PROGRAM MotionControl_sfc
VAR
	mcPower : MC_Power;
	mcSetPosition: MC_SetPosition;
	mcMoveAboslute: MC_MoveAbsolute;
	mcMoveRelative: MC_MoveRelative;
	mcMoveVelocity: MC_MoveVelocity;
	mcReset:MC_Reset;
	mcHalt:MC_Halt;
	mcStop:MC_Stop;
	
	bEnable : BOOL;
	bExecute_SPOS :BOOL;
	bExecute_MABS :BOOL;
	bExecute_MREL :BOOL;
	bExecute_RES :BOOL;
	bExecute_VEL :BOOL;
	bExecute_HALT :BOOL;
	bExecute_STOP :BOOL;
	
	fVelocity:LREAL;
	fPosition:LREAL;
	
	
	fAccel:LREAL;
END_VAR
VAR // added by the converter: edge detectors and wires of the graphical bodies
    _w1 : ANY;
END_VAR

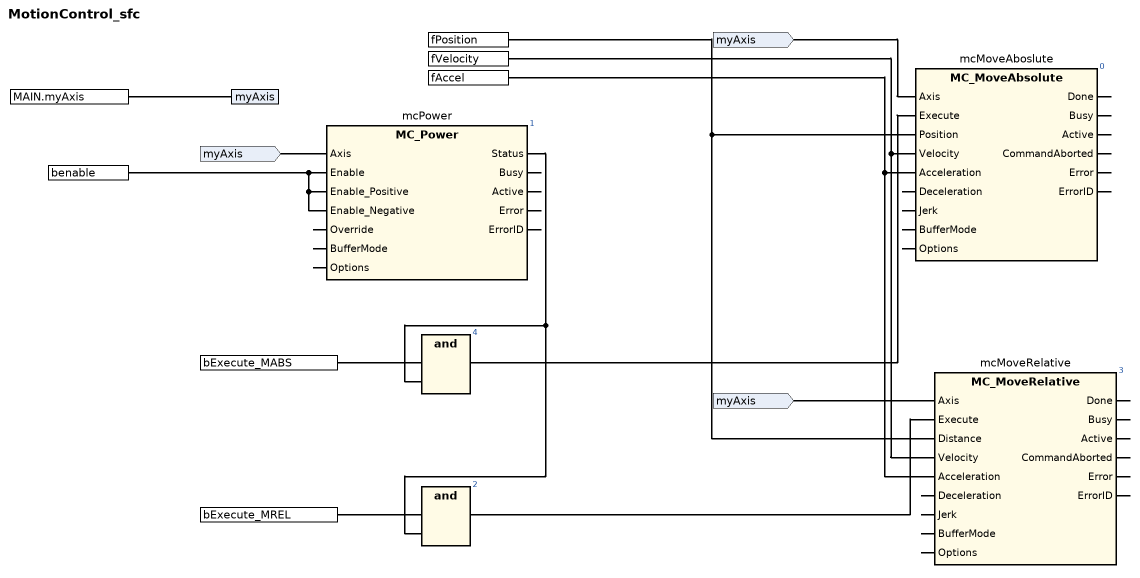
mcMoveAboslute(
    Axis := MAIN.myAxis,
    Execute := _w1,
    Position := fPosition,
    Velocity := fVelocity,
    Acceleration := fAccel); // MC_MoveAbsolute
mcPower(Axis := MAIN.myAxis, Enable := benable, Enable_Positive := benable, Enable_Negative := benable); // MC_Power
mcMoveRelative(
    Axis := MAIN.myAxis,
    Execute := bExecute_MREL AND mcPower.Status,
    Distance := fPosition,
    Velocity := fVelocity,
    Acceleration := fAccel); // MC_MoveRelative
_w1 := bExecute_MABS AND mcPower.Status;

END_PROGRAM

(* stored: Version 1.1.0.1, ProductVersion 3.1.4024.12
   POU MotionControl_sfc: Id {092693d0-e222-4c54-bdc4-611e5c46291f}, SpecialFunc None *)
